PROGRAM PRG_LVCP5_Colors
VAR
	arrLine : ARRAY[1..4] OF E_LineColors;
	arrCapacitorSchemaColor : ARRAY[1..7] OF ST_CapacitorSchemaColorWithContactor;

	i : INT;
	bInitDone : BOOL;
END_VAR

IF NOT bInitDone THEN
	ACT_ContactorConfigurations();
	bInitDone := TRUE;
END_IF

//line1
arrLine[1] := E_LineColors.Energised_Red;

//line2
arrLine[2] := arrLine[1];

//line3
arrLine[3] := arrLine[2];

//line4
arrLine[4] := arrLine[3];

//şemaları kendi içerisinde kontrol edicez
FOR i:=1 TO 10 DO
	arrCapacitorSchemaColor[i].GroundColor := E_LineColors.Grounded_Green;
	arrCapacitorSchemaColor[i].BottomLineColor2 := E_LineColors.Grounded_Green;

	//topline
	arrCapacitorSchemaColor[i].TopLineColor := arrLine[4];
	
	//bottomLine - şema üzerinde ayırıcının altındaki her iki line birbiri ile bağlantılı olduğu için tek yerden yönetiliyor
	IF arrCapacitorSchemaColor[i].ContactorPosition = E_ContactorPosition.ON THEN
		arrCapacitorSchemaColor[i].BottomLineColor := arrCapacitorSchemaColor[i].TopLineColor;
	ELSE
		arrCapacitorSchemaColor[i].BottomLineColor := E_LineColors.Default;
	END_IF
	
	//capacitor
	arrCapacitorSchemaColor[i].CapacitorColor := arrCapacitorSchemaColor[i].BottomLineColor;
	
END_FOR

ACTION ACT_ContactorConfigurations:
arrCapacitorSchemaColor[1].ContactorPosition := GVL_LVCP5.stGroup1_ContactorHMI.stStatus.ePosition;
arrCapacitorSchemaColor[2].ContactorPosition := GVL_LVCP5.stGroup2_ContactorHMI.stStatus.ePosition;
arrCapacitorSchemaColor[3].ContactorPosition := GVL_LVCP5.stGroup3_ContactorHMI.stStatus.ePosition;
arrCapacitorSchemaColor[4].ContactorPosition := GVL_LVCP5.stGroup4_ContactorHMI.stStatus.ePosition;
arrCapacitorSchemaColor[5].ContactorPosition := GVL_LVCP5.stGroup5_ContactorHMI.stStatus.ePosition;
arrCapacitorSchemaColor[6].ContactorPosition := GVL_LVCP5.stGroup6_ContactorHMI.stStatus.ePosition;
arrCapacitorSchemaColor[7].ContactorPosition := GVL_LVCP5.stGroup7_ContactorHMI.stStatus.ePosition;
END_ACTION

END_PROGRAM

(* stored: Version 1.1.0.1, ProductVersion 3.1.4024.13
   POU PRG_LVCP5_Colors: Id {2b6ced9f-e3a9-4282-a581-8d898f4977b9}, SpecialFunc None
   Action ACT_ContactorConfigurations: Id {b1067da9-a8b7-450d-9047-6bfae813f276} *)
